	    #actual^.vibrationSensor[0].i := 24;
	    #actual^.vibrationSensor[#actual^.vibrationSensor[0].i].scale.setInputMin := 0;
	    #actual^.vibrationSensor[#actual^.vibrationSensor[0].i].scale.setInputMax := 27600;
	    #actual^.vibrationSensor[#actual^.vibrationSensor[0].i].scale.setScaleMin := 0;
	    #actual^.vibrationSensor[#actual^.vibrationSensor[0].i].scale.setScaleMax := 250;//0 a 25mm
	    #actual^.vibrationSensor[#actual^.vibrationSensor[0].i].scale.setSignal :=
	    "=ecoat-32S2";//SENSOR DE VIBRAÇÃO BOMBA ULTRA-FILTRAÇÃO
	    "fScale"(#actual^.vibrationSensor[#actual^.vibrationSensor[0].i].scale);
	    #actual^.vibrationSensor[#actual^.vibrationSensor[0].i].signal :=
	    REAL_TO_INT(#actual^.vibrationSensor[#actual^.vibrationSensor[0].i].scale.getResult);

	    #actual^.vibrationSensor[0].i := 25;
	    #actual^.vibrationSensor[#actual^.vibrationSensor[0].i].scale.setInputMin := 0;
	    #actual^.vibrationSensor[#actual^.vibrationSensor[0].i].scale.setInputMax := 27600;
	    #actual^.vibrationSensor[#actual^.vibrationSensor[0].i].scale.setScaleMin := 0;
	    #actual^.vibrationSensor[#actual^.vibrationSensor[0].i].scale.setScaleMax := 250;//0 a 25mm
	    #actual^.vibrationSensor[#actual^.vibrationSensor[0].i].scale.setSignal :=
	    "=pre-55S1";//SENSOR DE VIBRAÇÃO BOMBA CIRCULAÇÃO REDE AGUA AQUECIDA BOILER ERZ900
	    "fScale"(#actual^.vibrationSensor[#actual^.vibrationSensor[0].i].scale);
	    #actual^.vibrationSensor[#actual^.vibrationSensor[0].i].signal :=
	    REAL_TO_INT(#actual^.vibrationSensor[#actual^.vibrationSensor[0].i].scale.getResult);
	END_REGION
	REGION conductivitySensor
	    #actual^.conductivitySensor[0].i := 1;
	    #actual^.conductivitySensor[#actual^.conductivitySensor[0].i].scale.setInputMin := 0;
	    #actual^.conductivitySensor[#actual^.conductivitySensor[0].i].scale.setInputMax := 27600;
	    #actual^.conductivitySensor[#actual^.conductivitySensor[0].i].scale.setScaleMin := 0;
	    #actual^.conductivitySensor[#actual^.conductivitySensor[0].i].scale.setScaleMax := 100;//ph
	    #actual^.conductivitySensor[#actual^.conductivitySensor[0].i].scale.setSignal :=
	    "=pre-56W1";//MEDIÇÃO DE CONDUTIVIDADE TANQUE AGUA D.I.
	    "fScale"(#actual^.conductivitySensor[#actual^.conductivitySensor[0].i].scale);
	    #actual^.conductivitySensor[#actual^.conductivitySensor[0].i].signal :=
	    REAL_TO_INT(#actual^.conductivitySensor[#actual^.conductivitySensor[0].i].scale.getResult);

	    #actual^.conductivitySensor[0].i := 7;
	    #actual^.conductivitySensor[#actual^.conductivitySensor[0].i].scale.setInputMin := 0;
	    #actual^.conductivitySensor[#actual^.conductivitySensor[0].i].scale.setInputMax := 27000;
	    #actual^.conductivitySensor[#actual^.conductivitySensor[0].i].scale.setScaleMin := 0;
	    #actual^.conductivitySensor[#actual^.conductivitySensor[0].i].scale.setScaleMax := 1000;//mS
	    #actual^.conductivitySensor[#actual^.conductivitySensor[0].i].scale.setSignal :=
	    "=pre-55F3";//MEDIÇÃO DE CONDUTIVIDADE TANQUE 07 ENXAGUE
	    "fScale"(#actual^.conductivitySensor[#actual^.conductivitySensor[0].i].scale);
	    #actual^.conductivitySensor[#actual^.conductivitySensor[0].i].signal :=
	    REAL_TO_INT(#actual^.conductivitySensor[#actual^.conductivitySensor[0].i].scale.getResult);

	    #actual^.conductivitySensor[0].i := 23;
	    #actual^.conductivitySensor[#actual^.conductivitySensor[0].i].scale.setInputMin := 0;
	    #actual^.conductivitySensor[#actual^.conductivitySensor[0].i].scale.setInputMax := 26900;
	    #actual^.conductivitySensor[#actual^.conductivitySensor[0].i].scale.setScaleMin := 0;
	    #actual^.conductivitySensor[#actual^.conductivitySensor[0].i].scale.setScaleMax := 10000; //mS
	    #actual^.conductivitySensor[#actual^.conductivitySensor[0].i].scale.setSignal :=
	    "=ecoat-34F1";//MEDIÇÃO DE CONDUTIVIDADE TANQUE 23 ANOLITO
	    "fScale"(#actual^.conductivitySensor[#actual^.conductivitySensor[0].i].scale);
	    #actual^.conductivitySensor[#actual^.conductivitySensor[0].i].signal :=
	    REAL_TO_INT(#actual^.conductivitySensor[#actual^.conductivitySensor[0].i].scale.getResult);
	END_REGION
	REGION phMeter
	    #actual^.phMeter[0].i := 11;
	    #actual^.phMeter[#actual^.phMeter[0].i].scale.setInputMin := 0;
	    #actual^.phMeter[#actual^.phMeter[0].i].scale.setInputMax := 27600;
	    #actual^.phMeter[#actual^.phMeter[0].i].scale.setScaleMin := 0;
	    #actual^.phMeter[#actual^.phMeter[0].i].scale.setScaleMax := 140;//ph
	    #actual^.phMeter[#actual^.phMeter[0].i].scale.setSignal :=
	    "=pre-55F2";//MEDIÇÃO DE PH TANQUE 11 NANOCERAMICO
	    "fScale"(#actual^.phMeter[#actual^.phMeter[0].i].scale);
	    #actual^.phMeter[#actual^.phMeter[0].i].signal :=
	    REAL_TO_INT(#actual^.phMeter[#actual^.phMeter[0].i].scale.getResult);

	    #actual^.phMeter[0].i := 13;
	    #actual^.phMeter[#actual^.phMeter[0].i].scale.setInputMin := 0;
	    #actual^.phMeter[#actual^.phMeter[0].i].scale.setInputMax := 27600;
	    #actual^.phMeter[#actual^.phMeter[0].i].scale.setScaleMin := 0;
	    #actual^.phMeter[#actual^.phMeter[0].i].scale.setScaleMax := 140;//ph
	    #actual^.phMeter[#actual^.phMeter[0].i].scale.setSignal :=
	    "=pre-55F1";//MEDIÇÃO DE PH TANQUE 08 NEUTRALIZADOR
	    "fScale"(#actual^.phMeter[#actual^.phMeter[0].i].scale);
	    #actual^.phMeter[#actual^.phMeter[0].i].signal :=
	    REAL_TO_INT(#actual^.phMeter[#actual^.phMeter[0].i].scale.getResult);
	END_REGION
	REGION flowIndicator
	    #actual^.flowIndicator[0].i += 1;
	    #actual^.flowIndicator[#actual^.flowIndicator[0].i].signal :=
	    "=ecoat-39S5:3"; //FLUXOSTATO SEGURANÇA BOMBA TRANSFERÊNCIA
	END_REGION
	REGION electricCurrent tank
	    #actual^.electricCurrent[0].i += 1;
	    #actual^.electricCurrent[#actual^.electricCurrent[0].i].scale.setSignal :=
	    "=ecoat-35W1";//MEDIÇÃO DE CORRENTE RETIFICADOR TANQUE 14 TINTA KTL
	    #actual^.electricCurrent[#actual^.electricCurrent[0].i].scale.setInputMin := 0;
	    #actual^.electricCurrent[#actual^.electricCurrent[0].i].scale.setInputMax := 28000;
	    #actual^.electricCurrent[#actual^.electricCurrent[0].i].scale.setScaleMin := 0;
	    #actual^.electricCurrent[#actual^.electricCurrent[0].i].scale.setScaleMax := 600;
	    "fScale"(#actual^.electricCurrent[#actual^.electricCurrent[0].i].scale);

	    #actual^.electricCurrent[0].i += 1;
	    #actual^.electricCurrent[#actual^.electricCurrent[0].i].scale.setSignal :=
	    "=ecoat-ecoatTensaoRetificador";//
	    #actual^.electricCurrent[#actual^.electricCurrent[0].i].scale.setInputMin := 0;
	    #actual^.electricCurrent[#actual^.electricCurrent[0].i].scale.setInputMax := 28000;
	    #actual^.electricCurrent[#actual^.electricCurrent[0].i].scale.setScaleMin := 0;
	    #actual^.electricCurrent[#actual^.electricCurrent[0].i].scale.setScaleMax := 512;
	    "fScale"(#actual^.electricCurrent[#actual^.electricCurrent[0].i].scale);

	END_REGION
	REGION consumptionMeter
	    #actual^.consumptionMeter[0].i += 1;
	    #actual^.consumptionMeter[#actual^.consumptionMeter[0].i].signal :=
	    "=pre-64S2:HF";//SINAL DE PULSO "A";MEDIDOR CONSUMO DE GÁS
	    #actual^.consumptionMeter[0].i += 1;
	    #actual^.consumptionMeter[#actual^.consumptionMeter[0].i].signal :=
	    "=pre-64S2:LF";//SINAL DE PULSO "B";MEDIDOR CONSUMO DE GÁS
	    #actual^.consumptionMeter[0].i += 1;
	    #actual^.consumptionMeter[#actual^.consumptionMeter[0].i].signal :=
	    "=pre-64S1:HF";//SINAL DE PULSO "A";MEDIDOR CONSUMO DE ÁGUA INDUSTRIAL
	    #actual^.consumptionMeter[0].i += 1;
	    #actual^.consumptionMeter[#actual^.consumptionMeter[0].i].signal :=
	    "=pre-64S1:LF";//SINAL DE PULSO "B";MEDIDOR CONSUMO DE ÁGUA INDUSTRIAL
	END_REGION
	REGION eom regular inputs
	    #actual^.confirmSetupTranslation[0].i += 1;
	    #actual^.confirmSetupTranslation[#actual^.confirmSetupTranslation[0].i].signal :=
	    "=eom01-7u1:Y2:Y13:3";//CONFIRMA SETUP MOVIMENTAÇÃO TRANSLAÇÃO  confirmSetupTranslation
	    #actual^.confirmSetupTranslation[0].i += 1;
	    #actual^.confirmSetupTranslation[#actual^.confirmSetupTranslation[0].i].signal :=
	    "=eom02-7u1:Y2:Y13:3";//CONFIRMA SETUP MOVIMENTAÇÃO TRANSLAÇÃO
	    #actual^.confirmSetupTranslation[0].i += 1;
	    #actual^.confirmSetupTranslation[#actual^.confirmSetupTranslation[0].i].signal :=
	    "=eom03-7u1:Y2:Y13:3";//CONFIRMA SETUP MOVIMENTAÇÃO TRANSLAÇÃO
	    #actual^.confirmSetupTranslation[0].i += 1;
	    #actual^.confirmSetupTranslation[#actual^.confirmSetupTranslation[0].i].signal :=
	    "=eom04-7u1:Y2:Y13:3";//CONFIRMA SETUP MOVIMENTAÇÃO TRANSLAÇÃO
	    #actual^.confirmSetupTranslation[0].i += 1;
	    #actual^.confirmSetupTranslation[#actual^.confirmSetupTranslation[0].i].signal :=
	    "=eom05-7u1:Y2:Y13:3";//CONFIRMA SETUP MOVIMENTAÇÃO TRANSLAÇÃO

	    #actual^.confirmTriggerGearmotorLift[0].i += 1;
	    #actual^.confirmTriggerGearmotorLift[#actual^.confirmTriggerGearmotorLift[0].i].signal :=
	    "=eom01-11k1:14";//CONFIRMA ACIONAMENTO MOTOREDUTOR ELEVAÇÃO  confirmTriggerGearmotorLift
	    #actual^.confirmTriggerGearmotorLift[0].i += 1;
	    #actual^.confirmTriggerGearmotorLift[#actual^.confirmTriggerGearmotorLift[0].i].signal :=
	    "=eom02-11k1:14";//CONFIRMA ACIONAMENTO MOTOREDUTOR ELEVAÇÃO
	    #actual^.confirmTriggerGearmotorLift[0].i += 1;
	    #actual^.confirmTriggerGearmotorLift[#actual^.confirmTriggerGearmotorLift[0].i].signal :=
	    "=eom03-11k1:14";//CONFIRMA ACIONAMENTO MOTOREDUTOR ELEVAÇÃO
	    #actual^.confirmTriggerGearmotorLift[0].i += 1;
	    #actual^.confirmTriggerGearmotorLift[#actual^.confirmTriggerGearmotorLift[0].i].signal :=
	    "=eom04-11k1:14";//CONFIRMA ACIONAMENTO MOTOREDUTOR ELEVAÇÃO
	    #actual^.confirmTriggerGearmotorLift[0].i += 1;
	    #actual^.confirmTriggerGearmotorLift[#actual^.confirmTriggerGearmotorLift[0].i].signal :=
	    "=eom05-11k1:14";//CONFIRMA ACIONAMENTO MOTOREDUTOR ELEVAÇÃO


	    #actual^.confirmTriggerGearmotorTranslation[0].i += 1;
	    #actual^.confirmTriggerGearmotorTranslation[#actual^.confirmTriggerGearmotorTranslation[0].i].signal :=
	    "=eom01-11k2:14";//CONFIRMA ACIONAMENTO MOTOREDUTOR TRANSLAÇÃO    confirmTriggerGearmotorTranslation
	    #actual^.confirmTriggerGearmotorTranslation[0].i += 1;
	    #actual^.confirmTriggerGearmotorTranslation[#actual^.confirmTriggerGearmotorTranslation[0].i].signal :=
	    "=eom02-11k2:14";//CONFIRMA ACIONAMENTO MOTOREDUTOR TRANSLAÇÃO
	    #actual^.confirmTriggerGearmotorTranslation[0].i += 1;
	    #actual^.confirmTriggerGearmotorTranslation[#actual^.confirmTriggerGearmotorTranslation[0].i].signal :=
	    "=eom03-11k2:14";//CONFIRMA ACIONAMENTO MOTOREDUTOR TRANSLAÇÃO
	    #actual^.confirmTriggerGearmotorTranslation[0].i += 1;
	    #actual^.confirmTriggerGearmotorTranslation[#actual^.confirmTriggerGearmotorTranslation[0].i].signal :=
	    "=eom04-11k2:14";//CONFIRMA ACIONAMENTO MOTOREDUTOR TRANSLAÇÃO
	    #actual^.confirmTriggerGearmotorTranslation[0].i += 1;
	    #actual^.confirmTriggerGearmotorTranslation[#actual^.confirmTriggerGearmotorTranslation[0].i].signal :=
	    "=eom05-11k2:14";//CONFIRMA ACIONAMENTO MOTOREDUTOR TRANSLAÇÃO

	    #actual^.minimumSafetyTranslation[0].i += 1;
	    #actual^.minimumSafetyTranslation[#actual^.minimumSafetyTranslation[0].i].signal :=
	    "=eom01-12b6:4";//LIMITE DE SEGURANÇA MÍNIMO MOVIMENTAÇÃO TRANSLAÇÃO    minimumSafetyTranslation
	    #actual^.minimumSafetyTranslation[0].i += 1;
	    #actual^.minimumSafetyTranslation[#actual^.minimumSafetyTranslation[0].i].signal :=
	    "=eom02-12b6:4";//LIMITE DE SEGURANÇA MÍNIMO MOVIMENTAÇÃO TRANSLAÇÃO
	    #actual^.minimumSafetyTranslation[0].i += 1;
	    #actual^.minimumSafetyTranslation[#actual^.minimumSafetyTranslation[0].i].signal :=
	    "=eom03-12b6:4";//LIMITE DE SEGURANÇA MÍNIMO MOVIMENTAÇÃO TRANSLAÇÃO
	    #actual^.minimumSafetyTranslation[0].i += 1;
	    #actual^.minimumSafetyTranslation[#actual^.minimumSafetyTranslation[0].i].signal :=
	    "=eom04-12b6:4";//LIMITE DE SEGURANÇA MÍNIMO MOVIMENTAÇÃO TRANSLAÇÃO
	    #actual^.minimumSafetyTranslation[0].i += 1;
	    #actual^.minimumSafetyTranslation[#actual^.minimumSafetyTranslation[0].i].signal :=
	    "=eom05-12b6:4";//LIMITE DE SEGURANÇA MÍNIMO MOVIMENTAÇÃO TRANSLAÇÃO


	    #actual^.safetyCrashCar[0].i += 1;
	    #actual^.safetyCrashCar[#actual^.safetyCrashCar[0].i].signal :=
	    "=eom01-12b7:4";//SEGURANCA COLISAO ENTRE CARROS DE TRANSFERENCIA   SafetyCrashCar
	    #actual^.safetyCrashCar[0].i += 1;
	    #actual^.safetyCrashCar[#actual^.safetyCrashCar[0].i].signal :=
	    "=eom02-12b7:4";//SEGURANCA COLISAO ENTRE CARROS DE TRANSFERENCIA
	    #actual^.safetyCrashCar[0].i += 1;
	    #actual^.safetyCrashCar[#actual^.safetyCrashCar[0].i].signal :=
	    "=eom03-12b7:4";//SEGURANCA COLISAO ENTRE CARROS DE TRANSFERENCIA
	    #actual^.safetyCrashCar[0].i += 1;
	    #actual^.safetyCrashCar[#actual^.safetyCrashCar[0].i].signal :=
	    "=eom04-12b7:4"; //SEGURANCA COLISAO ENTRE CARROS DE TRANSFERENCIA
	    #actual^.safetyCrashCar[0].i += 1;
	    #actual^.safetyCrashCar[#actual^.safetyCrashCar[0].i].signal :=
	    "=eom05-12b7:4";//SEGURANCA COLISAO ENTRE CARROS DE TRANSFERENCIA

	    #actual^.maximumSafetyTranslation[0].i += 1;
	    #actual^.maximumSafetyTranslation[#actual^.maximumSafetyTranslation[0].i].signal :=
	    "=eom01-13b4:4";//LIMITE DE SEGURANÇA MÁXIMO MOVIMENTAÇÃO TRANSLAÇÃO  maximumSafetyTranslation
	    #actual^.maximumSafetyTranslation[0].i += 1;
	    #actual^.maximumSafetyTranslation[#actual^.maximumSafetyTranslation[0].i].signal :=
	    "=eom02-13b4:4";//LIMITE DE SEGURANÇA MÁXIMO MOVIMENTAÇÃO TRANSLAÇÃO
	    #actual^.maximumSafetyTranslation[0].i += 1;
	    #actual^.maximumSafetyTranslation[#actual^.maximumSafetyTranslation[0].i].signal :=
	    "=eom03-13b4:4";//LIMITE DE SEGURANÇA MÁXIMO MOVIMENTAÇÃO TRANSLAÇÃO
	    #actual^.maximumSafetyTranslation[0].i += 1;
	    #actual^.maximumSafetyTranslation[#actual^.maximumSafetyTranslation[0].i].signal :=
	    "=eom04-13b4:4";//LIMITE DE SEGURANÇA MÁXIMO MOVIMENTAÇÃO TRANSLAÇÃO
	    #actual^.maximumSafetyTranslation[0].i += 1;
	    #actual^.maximumSafetyTranslation[#actual^.maximumSafetyTranslation[0].i].signal :=
	    "=eom05-13b4:4";//LIMITE DE SEGURANÇA MÁXIMO MOVIMENTAÇÃO TRANSLAÇÃO

	    #actual^.slowdownGoTranslation[0].i += 1;
	    #actual^.slowdownGoTranslation[#actual^.slowdownGoTranslation[0].i].signal :=
	    "=eom01-xed:8(1)";//DESACELERA MOVIMENTAÇÃO AVANÇO TRANSLAÇÃO     slowdownGoTranslation
	    #actual^.slowdownGoTranslation[0].i += 1;
	    #actual^.slowdownGoTranslation[#actual^.slowdownGoTranslation[0].i].signal :=
	    "=eom02-xed:8(1)";//DESACELERA MOVIMENTAÇÃO AVANÇO TRANSLAÇÃO
	    #actual^.slowdownGoTranslation[0].i += 1;
	    #actual^.slowdownGoTranslation[#actual^.slowdownGoTranslation[0].i].signal :=
	    "=eom03-xed:8(1)";//DESACELERA MOVIMENTAÇÃO AVANÇO TRANSLAÇÃO
	    #actual^.slowdownGoTranslation[0].i += 1;
	    #actual^.slowdownGoTranslation[#actual^.slowdownGoTranslation[0].i].signal :=
	    "=eom04-xed:8(1)";//DESACELERA MOVIMENTAÇÃO AVANÇO TRANSLAÇÃO
	    #actual^.slowdownGoTranslation[0].i += 1;
	    #actual^.slowdownGoTranslation[#actual^.slowdownGoTranslation[0].i].signal :=
	    "=eom05-xed:8(1)";//DESACELERA MOVIMENTAÇÃO AVANÇO TRANSLAÇÃO


	    #actual^.slowdownBackTranslation[0].i += 1;
	    #actual^.slowdownBackTranslation[#actual^.slowdownBackTranslation[0].i].status.setConfig := 0;
	    #actual^.slowdownBackTranslation[#actual^.slowdownBackTranslation[0].i].status.setDelayUp := 0;
	    #actual^.slowdownBackTranslation[#actual^.slowdownBackTranslation[0].i].status.setDelayDown := 50;
	    #actual^.slowdownBackTranslation[#actual^.slowdownBackTranslation[0].i].status.setSignal :=
	    "=eom01-xed:10";//DESACELERA MOVIMENTAÇÃO RECUO TRANSLAÇÃO    slowdownBackTranslation
	    "fStatus"(#actual^.slowdownBackTranslation[#actual^.slowdownBackTranslation[0].i].status);
	    #actual^.slowdownBackTranslation[#actual^.slowdownBackTranslation[0].i].signal :=
	    #actual^.slowdownBackTranslation[#actual^.slowdownBackTranslation[0].i].status.getStatus;
	    #actual^.slowdownBackTranslation[0].i += 1;
	    #actual^.slowdownBackTranslation[#actual^.slowdownBackTranslation[0].i].signal :=
	    "=eom02-xed:10";//DESACELERA MOVIMENTAÇÃO RECUO TRANSLAÇÃO
	    #actual^.slowdownBackTranslation[0].i += 1;
	    #actual^.slowdownBackTranslation[#actual^.slowdownBackTranslation[0].i].signal :=
	    "=eom03-xed:10";//DESACELERA MOVIMENTAÇÃO RECUO TRANSLAÇÃO
	    #actual^.slowdownBackTranslation[0].i += 1;
	    #actual^.slowdownBackTranslation[#actual^.slowdownBackTranslation[0].i].signal :=
	    "=eom04-xed:10";//DESACELERA MOVIMENTAÇÃO RECUO TRANSLAÇÃO
	    #actual^.slowdownBackTranslation[0].i += 1;
	    #actual^.slowdownBackTranslation[#actual^.slowdownBackTranslation[0].i].signal :=
	    "=eom05-xed:10";//DESACELERA MOVIMENTAÇÃO RECUO TRANSLAÇÃO

	    #actual^.positionStopTranslationTank[0].i += 1;
	    #actual^.positionStopTranslationTank[#actual^.positionStopTranslationTank[0].i].status.setConfig := 0;
	    #actual^.positionStopTranslationTank[#actual^.positionStopTranslationTank[0].i].status.setDelayUp := 0;
	    #actual^.positionStopTranslationTank[#actual^.positionStopTranslationTank[0].i].status.setDelayDown := 250;
	    #actual^.positionStopTranslationTank[#actual^.positionStopTranslationTank[0].i].status.setSignal :=
	    "=eom01-xed:9";//POSIÇÃO DE PARADA MOVIMENTAÇÃO TRANSLAÇÃO SOBRE O TANQUE   positionStopTranslationTank
	    "fStatus"(#actual^.positionStopTranslationTank[#actual^.positionStopTranslationTank[0].i].status);
	    #actual^.positionStopTranslationTank[#actual^.positionStopTranslationTank[0].i].signal :=
	    #actual^.positionStopTranslationTank[#actual^.positionStopTranslationTank[0].i].status.getStatus;

	    #actual^.positionStopTranslationTank[0].i += 1;
	    #actual^.positionStopTranslationTank[#actual^.positionStopTranslationTank[0].i].status.setConfig := 0;
	    #actual^.positionStopTranslationTank[#actual^.positionStopTranslationTank[0].i].status.setDelayUp := 0;
	    #actual^.positionStopTranslationTank[#actual^.positionStopTranslationTank[0].i].status.setDelayDown := 250;
	    #actual^.positionStopTranslationTank[#actual^.positionStopTranslationTank[0].i].status.setSignal :=
	    "=eom02-xed:9";//POSIÇÃO DE PARADA MOVIMENTAÇÃO TRANSLAÇÃO SOBRE O TANQUE   positionStopTranslationTank
	    "fStatus"(#actual^.positionStopTranslationTank[#actual^.positionStopTranslationTank[0].i].status);
	    #actual^.positionStopTranslationTank[#actual^.positionStopTranslationTank[0].i].signal :=
	    #actual^.positionStopTranslationTank[#actual^.positionStopTranslationTank[0].i].status.getStatus;

	    #actual^.positionStopTranslationTank[0].i += 1;
	    #actual^.positionStopTranslationTank[#actual^.positionStopTranslationTank[0].i].status.setConfig := 0;
	    #actual^.positionStopTranslationTank[#actual^.positionStopTranslationTank[0].i].status.setDelayUp := 0;
	    #actual^.positionStopTranslationTank[#actual^.positionStopTranslationTank[0].i].status.setDelayDown := 250;
	    #actual^.positionStopTranslationTank[#actual^.positionStopTranslationTank[0].i].status.setSignal :=
	    "=eom03-xed:9";//POSIÇÃO DE PARADA MOVIMENTAÇÃO TRANSLAÇÃO SOBRE O TANQUE   positionStopTranslationTank
	    "fStatus"(#actual^.positionStopTranslationTank[#actual^.positionStopTranslationTank[0].i].status);
	    #actual^.positionStopTranslationTank[#actual^.positionStopTranslationTank[0].i].signal :=
	    #actual^.positionStopTranslationTank[#actual^.positionStopTranslationTank[0].i].status.getStatus;

	    #actual^.positionStopTranslationTank[0].i += 1;
	    #actual^.positionStopTranslationTank[#actual^.positionStopTranslationTank[0].i].status.setConfig := 0;
	    #actual^.positionStopTranslationTank[#actual^.positionStopTranslationTank[0].i].status.setDelayUp := 0;
	    #actual^.positionStopTranslationTank[#actual^.positionStopTranslationTank[0].i].status.setDelayDown := 250;
	    #actual^.positionStopTranslationTank[#actual^.positionStopTranslationTank[0].i].status.setSignal :=
	    "=eom04-xed:9";//POSIÇÃO DE PARADA MOVIMENTAÇÃO TRANSLAÇÃO SOBRE O TANQUE   positionStopTranslationTank
	    "fStatus"(#actual^.positionStopTranslationTank[#actual^.positionStopTranslationTank[0].i].status);
	    #actual^.positionStopTranslationTank[#actual^.positionStopTranslationTank[0].i].signal :=
	    #actual^.positionStopTranslationTank[#actual^.positionStopTranslationTank[0].i].status.getStatus;

	    #actual^.positionStopTranslationTank[0].i += 1;
	    #actual^.positionStopTranslationTank[#actual^.positionStopTranslationTank[0].i].status.setConfig := 0;
	    #actual^.positionStopTranslationTank[#actual^.positionStopTranslationTank[0].i].status.setDelayUp := 0;
	    #actual^.positionStopTranslationTank[#actual^.positionStopTranslationTank[0].i].status.setDelayDown := 250;
	    #actual^.positionStopTranslationTank[#actual^.positionStopTranslationTank[0].i].status.setSignal :=
	    //"=eom05-XED:9";//POSIÇÃO DE PARADA MOVIMENTAÇÃO TRANSLAÇÃO SOBRE O TANQUE   positionStopTranslationTank
	    "=eom05-13b4:4" OR //LIMITE DE SEGURANÇA MÁXIMO MOVIMENTAÇÃO TRANSLAÇÃO
	    "=eom05-12b6:4";//LIMITE DE SEGURANÇA MÍNIMO MOVIMENTAÇÃO TRANSLAÇÃO
	    "fStatus"(#actual^.positionStopTranslationTank[#actual^.positionStopTranslationTank[0].i].status);
	    #actual^.positionStopTranslationTank[#actual^.positionStopTranslationTank[0].i].signal :=
	    #actual^.positionStopTranslationTank[#actual^.positionStopTranslationTank[0].i].status.getStatus;

	    #actual^.limitMaximumClimbLift[0].i += 1;
	    #actual^.limitMaximumClimbLift[#actual^.limitMaximumClimbLift[0].i].status.setConfig := 0;
	    #actual^.limitMaximumClimbLift[#actual^.limitMaximumClimbLift[0].i].status.setDelayUp := 250;
	    #actual^.limitMaximumClimbLift[#actual^.limitMaximumClimbLift[0].i].status.setDelayDown := 500;
	    #actual^.limitMaximumClimbLift[#actual^.limitMaximumClimbLift[0].i].status.setSignal :=
	    "=eom01-12b5:4";//LIMITE MÁXIMO DESLOCAMENTO SUBIDA DO ELEVADOR    limitMaximumClimbLift
	    "fStatus"(#actual^.limitMaximumClimbLift[#actual^.limitMaximumClimbLift[0].i].status);
	    #actual^.limitMaximumClimbLift[#actual^.limitMaximumClimbLift[0].i].signal :=
	    #actual^.limitMaximumClimbLift[#actual^.limitMaximumClimbLift[0].i].status.getStatus;

	    #actual^.limitMaximumClimbLift[0].i += 1;
	    #actual^.limitMaximumClimbLift[#actual^.limitMaximumClimbLift[0].i].status.setConfig := 0;
	    #actual^.limitMaximumClimbLift[#actual^.limitMaximumClimbLift[0].i].status.setDelayUp := 250;
	    #actual^.limitMaximumClimbLift[#actual^.limitMaximumClimbLift[0].i].status.setDelayDown := 500;
	    #actual^.limitMaximumClimbLift[#actual^.limitMaximumClimbLift[0].i].status.setSignal :=
	    "=eom02-12b5:4";//LIMITE MÁXIMO DESLOCAMENTO SUBIDA DO ELEVADOR
	    "fStatus"(#actual^.limitMaximumClimbLift[#actual^.limitMaximumClimbLift[0].i].status);
	    #actual^.limitMaximumClimbLift[#actual^.limitMaximumClimbLift[0].i].signal :=
	    #actual^.limitMaximumClimbLift[#actual^.limitMaximumClimbLift[0].i].status.getStatus;

	    #actual^.limitMaximumClimbLift[0].i += 1;
	    #actual^.limitMaximumClimbLift[#actual^.limitMaximumClimbLift[0].i].status.setConfig := 0;
	    #actual^.limitMaximumClimbLift[#actual^.limitMaximumClimbLift[0].i].status.setDelayUp := 250;
	    #actual^.limitMaximumClimbLift[#actual^.limitMaximumClimbLift[0].i].status.setDelayDown := 500;
	    #actual^.limitMaximumClimbLift[#actual^.limitMaximumClimbLift[0].i].status.setSignal :=
	    "=eom03-12b5:4";//LIMITE MÁXIMO DESLOCAMENTO SUBIDA DO ELEVADOR
	    "fStatus"(#actual^.limitMaximumClimbLift[#actual^.limitMaximumClimbLift[0].i].status);
	    #actual^.limitMaximumClimbLift[#actual^.limitMaximumClimbLift[0].i].signal :=
	    #actual^.limitMaximumClimbLift[#actual^.limitMaximumClimbLift[0].i].status.getStatus;

	    #actual^.limitMaximumClimbLift[0].i += 1;
	    #actual^.limitMaximumClimbLift[#actual^.limitMaximumClimbLift[0].i].status.setConfig := 0;
	    #actual^.limitMaximumClimbLift[#actual^.limitMaximumClimbLift[0].i].status.setDelayUp := 250;
	    #actual^.limitMaximumClimbLift[#actual^.limitMaximumClimbLift[0].i].status.setDelayDown := 500;
	    #actual^.limitMaximumClimbLift[#actual^.limitMaximumClimbLift[0].i].status.setSignal :=
	    "=eom04-12b5:4";//LIMITE MÁXIMO DESLOCAMENTO SUBIDA DO ELEVADOR
	    "fStatus"(#actual^.limitMaximumClimbLift[#actual^.limitMaximumClimbLift[0].i].status);
	    #actual^.limitMaximumClimbLift[#actual^.limitMaximumClimbLift[0].i].signal :=
	    #actual^.limitMaximumClimbLift[#actual^.limitMaximumClimbLift[0].i].status.getStatus;

	    #actual^.limitMaximumClimbLift[0].i += 1;
	    #actual^.limitMaximumClimbLift[#actual^.limitMaximumClimbLift[0].i].status.setConfig := 0;
	    #actual^.limitMaximumClimbLift[#actual^.limitMaximumClimbLift[0].i].status.setDelayUp := 250;
	    #actual^.limitMaximumClimbLift[#actual^.limitMaximumClimbLift[0].i].status.setDelayDown := 500;
	    #actual^.limitMaximumClimbLift[#actual^.limitMaximumClimbLift[0].i].status.setSignal :=
	    "=eom05-12b5:4";//LIMITE MÁXIMO DESLOCAMENTO SUBIDA DO ELEVADOR
	    "fStatus"(#actual^.limitMaximumClimbLift[#actual^.limitMaximumClimbLift[0].i].status);
	    #actual^.limitMaximumClimbLift[#actual^.limitMaximumClimbLift[0].i].signal :=
	    #actual^.limitMaximumClimbLift[#actual^.limitMaximumClimbLift[0].i].status.getStatus;

	    #actual^.slowdownClimbLift[0].i += 1;
	    #actual^.slowdownClimbLift[#actual^.slowdownClimbLift[0].i].signal :=
	    "=eom01-12b4:4";//DESACELERACAO DESLOCAMENTO SUBIDA DO ELEVADOR   slowdownClimbLift
	    #actual^.slowdownClimbLift[0].i += 1;
	    #actual^.slowdownClimbLift[#actual^.slowdownClimbLift[0].i].signal :=
	    "=eom02-12b4:4";//DESACELERACAO DESLOCAMENTO SUBIDA DO ELEVADOR
	    #actual^.slowdownClimbLift[0].i += 1;
	    #actual^.slowdownClimbLift[#actual^.slowdownClimbLift[0].i].signal :=
	    "=eom03-12b4:4";//DESACELERACAO DESLOCAMENTO SUBIDA DO ELEVADOR
	    #actual^.slowdownClimbLift[0].i += 1;
	    #actual^.slowdownClimbLift[#actual^.slowdownClimbLift[0].i].signal :=
	    "=eom04-12b4:4";//DESACELERACAO DESLOCAMENTO SUBIDA DO ELEVADOR
	    #actual^.slowdownClimbLift[0].i += 1;
	    #actual^.slowdownClimbLift[#actual^.slowdownClimbLift[0].i].signal :=
	    "=eom05-12b4:4";//DESACELERACAO DESLOCAMENTO SUBIDA DO ELEVADOR

	    #actual^.slowdownDescentLift[0].i += 1;
	    #actual^.slowdownDescentLift[#actual^.slowdownDescentLift[0].i].signal :=
	    "=eom01-12b3:4";//DESACELERACAO DESLOCAMENTO DESCIDA DO ELEVADOR      slowdownDescentLift
	    #actual^.slowdownDescentLift[0].i += 1;
	    #actual^.slowdownDescentLift[#actual^.slowdownDescentLift[0].i].signal :=
	    "=eom02-12b3:4";//DESACELERACAO DESLOCAMENTO DESCIDA DO ELEVADOR
	    #actual^.slowdownDescentLift[0].i += 1;
	    #actual^.slowdownDescentLift[#actual^.slowdownDescentLift[0].i].signal :=
	    "=eom03-12b3:4";//DESACELERACAO DESLOCAMENTO DESCIDA DO ELEVADOR
	    #actual^.slowdownDescentLift[0].i += 1;
	    #actual^.slowdownDescentLift[#actual^.slowdownDescentLift[0].i].signal :=
	    "=eom04-12b3:4";//DESACELERACAO DESLOCAMENTO DESCIDA DO ELEVADOR
	    #actual^.slowdownDescentLift[0].i += 1;
	    #actual^.slowdownDescentLift[#actual^.slowdownDescentLift[0].i].signal :=
	    "=eom05-12b3:4";//DESACELERACAO DESLOCAMENTO DESCIDA DO ELEVADOR

	    #actual^.limitMiddleDescentLift[0].i += 1;
	    #actual^.limitMiddleDescentLift[#actual^.limitMiddleDescentLift[0].i].signal :=
	    "=eom01-12b2:4";//LIMITE INTERMEDIÁRIO DESLOCAMENTO DESCIDA DO ELEVADOR   limitMiddleDescentLift
	    #actual^.limitMiddleDescentLift[0].i += 1;
	    #actual^.limitMiddleDescentLift[#actual^.limitMiddleDescentLift[0].i].signal :=
	    "=eom02-12b2:4";//LIMITE INTERMEDIÁRIO DESLOCAMENTO DESCIDA DO ELEVADOR
	    #actual^.limitMiddleDescentLift[0].i += 1;
	    #actual^.limitMiddleDescentLift[#actual^.limitMiddleDescentLift[0].i].signal :=
	    "=eom03-12b2:4";//LIMITE INTERMEDIÁRIO DESLOCAMENTO DESCIDA DO ELEVADOR
	    #actual^.limitMiddleDescentLift[0].i += 1;
	    #actual^.limitMiddleDescentLift[#actual^.limitMiddleDescentLift[0].i].signal :=
	    "=eom04-12b2:4";//LIMITE INTERMEDIÁRIO DESLOCAMENTO DESCIDA DO ELEVADOR
	    #actual^.limitMiddleDescentLift[0].i += 1;
	    #actual^.limitMiddleDescentLift[#actual^.limitMiddleDescentLift[0].i].signal :=
	    "=eom05-12b2:4";//LIMITE INTERMEDIÁRIO DESLOCAMENTO DESCIDA DO ELEVADOR

	    #actual^.limitMinimumDescentLift[0].i += 1;
	    #actual^.limitMinimumDescentLift[#actual^.limitMinimumDescentLift[0].i].signal :=
	    "=eom01-12b1:4";//LIMITE MÍNIMO DESLOCAMENTO DESCIDA DO ELEVADOR     LimitMinimumDescentLift
	    #actual^.limitMinimumDescentLift[0].i += 1;
	    #actual^.limitMinimumDescentLift[#actual^.limitMinimumDescentLift[0].i].signal :=
	    "=eom02-12b1:4";//LIMITE MÍNIMO DESLOCAMENTO DESCIDA DO ELEVADOR
	    #actual^.limitMinimumDescentLift[0].i += 1;
	    #actual^.limitMinimumDescentLift[#actual^.limitMinimumDescentLift[0].i].signal :=
	    "=eom03-12b1:4";//LIMITE MÍNIMO DESLOCAMENTO DESCIDA DO ELEVADOR
	    #actual^.limitMinimumDescentLift[0].i += 1;
	    #actual^.limitMinimumDescentLift[#actual^.limitMinimumDescentLift[0].i].signal :=
	    "=eom04-12b1:4";//LIMITE MÍNIMO DESLOCAMENTO DESCIDA DO ELEVADOR
	    #actual^.limitMinimumDescentLift[0].i += 1;
	    #actual^.limitMinimumDescentLift[#actual^.limitMinimumDescentLift[0].i].signal :=
	    "=eom05-12b1:4";//LIMITE MÍNIMO DESLOCAMENTO DESCIDA DO ELEVADOR

	    #actual^.proximitySensor[0].i += 1;
	    #actual^.proximitySensor[#actual^.proximitySensor[0].i].signal :=
	    FALSE; //SENSOR DE APROXIMAÇÃO
	    #actual^.proximitySensor[0].i += 1;
	    #actual^.proximitySensor[#actual^.proximitySensor[0].i].signal :=
	    "=eom02-aproxE2"; //SENSOR DE APROXIMAÇÃO
	    #actual^.proximitySensor[0].i += 1;
	    #actual^.proximitySensor[#actual^.proximitySensor[0].i].signal :=
	    "=eom03-aproxE3"; //SENSOR DE APROXIMAÇÃO
	    #actual^.proximitySensor[0].i += 1;
	    #actual^.proximitySensor[#actual^.proximitySensor[0].i].signal :=
	    "=eom04-aproxE4"; //SENSOR DE APROXIMAÇÃO

	END_REGION
	REGION conveyorEncoder
	    #actual^.conveyorEncoder[0].i += 4;
	    #autoConveyor := REF("dbArchiveAutoConveyor".autoConveyor[4]);
	    #control := REF("dbArchiveControlConveyor".controlConveyor[3].control[1]);
	    #actual^.conveyorEncoder[#actual^.conveyorEncoder[0].i].pulse.setSignal :=
	    "=oven-ovenCounter".%X10;
	    "fPulseOnRise"(#actual^.conveyorEncoder[#actual^.conveyorEncoder[0].i].pulse);

	    IF #actual^.conveyorEncoder[#actual^.conveyorEncoder[0].i].pulse.getSignal THEN
	        #control := REF("dbArchiveControlConveyor".controlConveyor[4].control[1]);
	        IF #control^.command.getTurnOnForward THEN
	            #actual^.conveyorEncoder[#actual^.conveyorEncoder[0].i].i += 1;
	        END_IF;
	        IF #control^.command.getTurnOnReturn THEN
	            #actual^.conveyorEncoder[#actual^.conveyorEncoder[0].i].i -= 1;
	        END_IF;
	    END_IF;

	    IF #actual^.conveyorEncoder[#actual^.conveyorEncoder[0].i].i > 156 OR
	        #actual^.conveyorEncoder[#actual^.conveyorEncoder[0].i].i < 1 THEN
	        #actual^.conveyorEncoder[#actual^.conveyorEncoder[0].i].i := 1;
	    END_IF;

	    #tempBool := FALSE;
	    FOR #ia := 1 TO 4 DO
	        #slot := REF("dbArchiveSlotConveyor".slotConveyor[4].slot[#ia]);
	        IF #slot^.info.data.getDataReady OR #slot^.info.data.getOccupied THEN
	            #tempBool := TRUE;
	        END_IF;
	    END_FOR;

	    IF NOT #tempBool THEN
	        #actual^.conveyorEncoder[#actual^.conveyorEncoder[0].i].i := 1;
	    END_IF;

	    IF (#actual^.skidDetectedFConveyor[3].pulse.getSignal AND #control^.command.getTurnOnForward) THEN
	        #actual^.conveyorEncoder[#actual^.conveyorEncoder[0].i].i := 120;
	    END_IF;

	    IF #actual^.conveyorEncoder[#actual^.conveyorEncoder[0].i].i >= 1 AND
	        #actual^.conveyorEncoder[#actual^.conveyorEncoder[0].i].i <= 98 THEN
	        #actual^.conveyorEncoder[#actual^.conveyorEncoder[0].i].signal := TRUE;
	    ELSE
	        #actual^.conveyorEncoder[#actual^.conveyorEncoder[0].i].signal := FALSE;
	    END_IF;


	    //
	    #actual^.conveyorEncoder[0].i += 2;
	    #autoConveyor := REF("dbArchiveAutoConveyor".autoConveyor[6]);
	    #control := REF("dbArchiveControlConveyor".controlConveyor[5].control[1]);
	    #slot := REF("dbArchiveSlotConveyor".slotConveyor[5].slot[1]);
	    #actual^.conveyorEncoder[#actual^.conveyorEncoder[0].i].pulse.setSignal :=
	    "=pre-preCounter".%X10;

	    IF #actual^.skidDetectedAConveyor[6].pulse.getSignal THEN
	        #actual^.conveyorEncoder[#actual^.conveyorEncoder[0].i].i := 150;
	    END_IF;

	    "fPulseOnRise"(#actual^.conveyorEncoder[#actual^.conveyorEncoder[0].i].pulse);
	    IF #actual^.conveyorEncoder[#actual^.conveyorEncoder[0].i].pulse.getSignal THEN
	        #control := REF("dbArchiveControlConveyor".controlConveyor[6].control[1]);
	        IF #control^.command.getTurnOnForward THEN
	            #actual^.conveyorEncoder[#actual^.conveyorEncoder[0].i].i += 1;
	        END_IF;
	        IF #control^.command.getTurnOnReturn THEN
	            #actual^.conveyorEncoder[#actual^.conveyorEncoder[0].i].i -= 1;
	        END_IF;
	    END_IF;

	    IF #actual^.conveyorEncoder[#actual^.conveyorEncoder[0].i].i > 156 OR
	        #actual^.conveyorEncoder[#actual^.conveyorEncoder[0].i].i < 1 THEN
	        #actual^.conveyorEncoder[#actual^.conveyorEncoder[0].i].i := 1;
	    END_IF;

	    IF #actual^.conveyorEncoder[#actual^.conveyorEncoder[0].i].i >= 1 AND
	        #actual^.conveyorEncoder[#actual^.conveyorEncoder[0].i].i <= 98 THEN
	        #actual^.conveyorEncoder[#actual^.conveyorEncoder[0].i].signal := TRUE;
	    ELSE
	        #actual^.conveyorEncoder[#actual^.conveyorEncoder[0].i].signal := FALSE;
	    END_IF;

	END_REGION
	REGION count qty
	    #tempInt := #actual^.circuitBreaker[0].i;
	    #tempInt := #actual^.resetFailure[0].i;
	    #tempInt := #actual^.minimumSafetyLevel[0].i;
	    #tempInt := #actual^.maximumSafetyLevel[0].i;
	    #tempInt := #actual^.maximumLevel[0].i;
	    #tempInt := #actual^.minimumLevel[0].i;
	    #tempInt := #actual^.returnedADoor[0].i;
	    #tempInt := #actual^.advancedADoor[0].i;
	    #tempInt := #actual^.returnedBDoor[0].i;
	    #tempInt := #actual^.advancedBDoor[0].i;
	    #tempInt := #actual^.temperatureOven[0].i;
	    #tempInt := #actual^.temperatureInBoiler[0].i;
	    #tempInt := #actual^.temperatureOutBoiler[0].i;
	    #tempInt := #actual^.temperatureTank[0].i;
	    #tempInt := #actual^.rightArrow[0].i;
	    #tempInt := #actual^.rightArrow[0].i;
	    #tempInt := #actual^.downArrow[0].i;
	    #tempInt := #actual^.upArrow[0].i;
	    #tempInt := #actual^.skidDetectedATank[0].i;
	    #tempInt := #actual^.skidDetectedAConveyor[0].i;
	    #tempInt := #actual^.skidDetectedAShipping[0].i;
	    #tempInt := #actual^.resetSafety[0].i;
	    #tempInt := #actual^.confirmSetupTranslation[0].i;
	    #tempInt := #actual^.confirmTriggerGearmotorLift[0].i;
	    #tempInt := #actual^.confirmTriggerGearmotorTranslation[0].i;
	    #tempInt := #actual^.slowdownDescentLift[0].i;
	    #tempInt := #actual^.slowdownClimbLift[0].i;
	    #tempInt := #actual^.slowdownGoTranslation[0].i;
	    #tempInt := #actual^.slowdownBackTranslation[0].i;
	    #tempInt := #actual^.positionStopTranslationTank[0].i;
	    #tempInt := #actual^.limitMinimumDescentLift[0].i;
	    #tempInt := #actual^.limitMaximumClimbLift[0].i;
	    #tempInt := #actual^.slowdownGoTranslation[0].i;
	    #tempInt := #actual^.slowdownBackTranslation[0].i;
	    #tempInt := #actual^.positionStopTranslationTank[0].i;
	    #tempInt := #actual^.limitMinimumDescentLift[0].i;
	    #tempInt := #actual^.limitMaximumClimbLift[0].i;
	    #tempInt := #actual^.limitMiddleDescentLift[0].i;
	    #tempInt := #actual^.maximumSafetyTranslation[0].i;
	    #tempInt := #actual^.minimumSafetyTranslation[0].i;
	    #tempInt := #actual^.safetyCrashCar[0].i;
	    #tempInt := #actual^.vibrationSensor[0].i;
	    #tempInt := #actual^.conductivitySensor[0].i;
	    #tempInt := #actual^.phMeter[0].i;
	    #tempInt := #actual^.heatingResistorFailure[0].i;
	    #tempInt := #actual^.burnerFailure[0].i;
	    #tempInt := #actual^.chillerFailure[0].i;
	    #tempInt := #actual^.skidDetectedBConveyor[0].i;
	    #tempInt := #actual^.skidDetectedCConveyor[0].i;
	    #tempInt := #actual^.skidDetectedDConveyor[0].i;
	    #tempInt := #actual^.skidDetectedEConveyor[0].i;
	    #tempInt := #actual^.skidDetectedFConveyor[0].i;
	    #tempInt := #actual^.skidDetectedBShipping[0].i;
	    #tempInt := #actual^.skidDetectedCShipping[0].i;
	    #tempInt := #actual^.eletronicCircuitBreaker[0].i;
	    #tempInt := #actual^.powerFailure[0].i;
	    #tempInt := #actual^."remote"[0].i;
	    #tempInt := #actual^.thermostatIndication[0].i;
	    #tempInt := #actual^.stopMotion[0].i;
	    #tempInt := #actual^.safetyContactorFeedback[0].i;
	    #tempInt := #actual^.pressureTransmitter[0].i;
	    #tempInt := #actual^.airConditioningFailure[0].i;
	    #tempInt := #actual^.flowIndicator[0].i;
	    #tempInt := #actual^.electricCurrent[0].i;
	    #tempInt := #actual^.advancedConveyor[0].i;
	    #tempInt := #actual^.returnedConveyor[0].i;
	    #tempInt := #actual^.consumptionMeter[0].i;
	    #tempInt := #actual^.resistorPowerController[0].i;
	    #tempInt := #actual^.remoteFastModeFR[0].i;
	    #tempInt := #actual^.remoteFastModeUD[0].i;
	    #tempInt := #actual^.netDiag[0].i;
	    #tempInt := #actual^.tankTelegramRecirculation[0].i;
	    #tempInt := #actual^.conveyorTelegram[0].i;
	    #tempInt := #actual^.doorTelegram[0].i;
	    #tempInt := #actual^.exhaustTelegram[0].i;
	    #tempInt := #actual^.proximitySensor[0].i;
	    #tempInt := #actual^.conveyorEncoder[0].i;
	END_REGION
	REGION global status
	    #actual^.generalResetFailure.signal := FALSE;
	    FOR #i := 1 TO #actual^.resetFailure[0].i DO
	        IF #actual^.resetFailure[#i].signal OR
	            "dbUtilities".autoReset.getStatus THEN
	            #actual^.generalResetFailure.signal := TRUE;
	        END_IF;
	    END_FOR;
	    #actual^.generalStopMotion.signal := FALSE;
	    FOR #i := 1 TO #actual^.stopMotion[0].i DO
	        IF NOT #actual^.stopMotion[#i].signal THEN
	            #actual^.generalStopMotion.signal := TRUE;
	        END_IF;
	    END_FOR;
	END_REGION
END_FUNCTION

